{attribute 'qualified_only'}
{attribute 'to_string'}
TYPE E_MoveState :
(
    IDLING:=0,
    INIT:=10,
    STARTED:=20,
    IN_PROGRESS :=30,
    REACHED:=40,
    INTERRUPTED:=50,
    DONE:=60,
    ERROR:=-99
) INT;
END_TYPE

(* stored: Version 1.1.0.1
   DUT E_MoveState: Id {933b85d6-53dd-4c3d-b3b1-3a89b00aa8fa} *)
